// TIA Portal V17 export
// export: Created 2025-03-05T08:02:23.2667087Z, ExportSetting WithDefaults, DisplayName Totally Integrated Automation Portal, DisplayVersion V17 Update 8, DisplayName TIA Portal Openness, DisplayVersion V17 Update 8, DisplayName TIA Portal Version Control Interface, DisplayVersion V17, DisplayName SINAMICS Startdrive Advanced, DisplayVersion V17 SP2, DisplayName SINAMICS Startdrive G110M, G120, G120C, G120D, G120P, G115D, DisplayVersion V17 SP2, DisplayName SINAMICS Startdrive G130, G150, S120, S150, SINAMICS MV, S210, DisplayVersion V17 SP2, DisplayName STEP 7 Professional, DisplayVersion V17 Update 8, DisplayName SINUMERIK ONE STEP 7 Toolbox, DisplayVersion V17 Update 12, DisplayName SINUMERIK 840D sl STEP 7 Toolbox, DisplayVersion V17 Update 12, DisplayName STEP 7 Safety, DisplayVersion V17 Update 6, DisplayName WinCC Advanced, DisplayVersion V17 Update 8
TYPE "LAYOUT"
// stored: IsFailsafeCompliant false
   STRUCT
      Arrow : Array[0..79] of Bool;   // Arrow
      LED : Array[0..79] of Bool;   // LED
      Image : Array[0..79] of Bool;   // Image
      Text : Array[0..79] of Bool;   // Text
      IO_field : Array[0..79] of Bool;   // IO_field
      ProgressBar : Array[0..79] of Bool;   // ProgressBar
      Table0 : Bool;   // Table0
      Table1 : Bool;   // Table1
      Table2 : Bool;   // Table2
      Table3 : Bool;   // Table3
      Table4 : Bool;   // Table4
      Table5 : Bool;   // Table5
      Table6 : Bool;   // Table6
      Table7 : Bool;   // Table7
      Curve0 : Bool;   // Curve0
      Curve1 : Bool;   // Curve1
      Curve2 : Bool;   // Curve2
      Curve3 : Bool;   // Curve3
      Curve4 : Bool;   // Curve4
      Curve5 : Bool;   // Curve5
      Curve6 : Bool;   // Curve6
      Curve7 : Bool;   // Curve7
      Internet0 : Bool;   // Internet0
      Internet1 : Bool;   // Internet1
      Internet2 : Bool;   // Internet2
      Internet3 : Bool;   // Internet3
      Internet4 : Bool;   // Internet4
      Internet5 : Bool;   // Internet5
      Internet6 : Bool;   // Internet6
      Internet7 : Bool;   // Internet7
      SoftkeyLeft0 : Bool;   // SoftkeyLeft0
      SoftkeyLeft1 : Bool;   // SoftkeyLeft1
      SoftkeyLeft2 : Bool;   // SoftkeyLeft2
      SoftkeyLeft3 : Bool;   // SoftkeyLeft3
      SoftkeyLeft4 : Bool;   // SoftkeyLeft4
      SoftkeyLeft5 : Bool;   // SoftkeyLeft5
      SoftkeyLeftAll : Bool;   // SoftkeyLeftAll
      reserveleft : Bool;   // reserveleft
      SoftkeyRight0 : Bool;   // SoftkeyRight0
      SoftkeyRight1 : Bool;   // SoftkeyRight1
      SoftkeyRight2 : Bool;   // SoftkeyRight2
      SoftkeyRight3 : Bool;   // SoftkeyRight3
      SoftkeyRight4 : Bool;   // SoftkeyRight4
      SoftkeyRight5 : Bool;   // SoftkeyRight5
      SoftkeyRightAll : Bool;   // SoftkeyRightAll
      reserveright : Bool;   // reserveright
      Pushbutton0 : Bool;   // Pushbutton0
      Pushbutton1 : Bool;   // Pushbutton1
      Pushbutton2 : Bool;   // Pushbutton2
      Pushbutton3 : Bool;   // Pushbutton3
      Pushbutton4 : Bool;   // Pushbutton4
      Pushbutton5 : Bool;   // Pushbutton5
      Pushbutton6 : Bool;   // Pushbutton6
      Pushbutton7 : Bool;   // Pushbutton7
      Pushbutton8 : Bool;   // Pushbutton8
      Pushbutton9 : Bool;   // Pushbutton9
      Pushbutton10 : Bool;   // Pushbutton10
      Pushbutton11 : Bool;   // Pushbutton11
      Pushbutton12 : Bool;   // Pushbutton12
      Pushbutton13 : Bool;   // Pushbutton13
      Pushbutton14 : Bool;   // Pushbutton14
      Pushbutton15 : Bool;   // Pushbutton15
      Pushbutton16 : Bool;   // Pushbutton16
      Pushbutton17 : Bool;   // Pushbutton17
      Pushbutton18 : Bool;   // Pushbutton18
      Pushbutton19 : Bool;   // Pushbutton19
      Pushbutton20 : Bool;   // Pushbutton20
      Pushbutton21 : Bool;   // Pushbutton21
      Pushbutton22 : Bool;   // Pushbutton22
      Pushbutton23 : Bool;   // Pushbutton23
      Pushbutton24 : Bool;   // Pushbutton24
      Pushbutton25 : Bool;   // Pushbutton25
      Pushbutton26 : Bool;   // Pushbutton26
      Pushbutton27 : Bool;   // Pushbutton27
      Pushbutton28 : Bool;   // Pushbutton28
      Pushbutton29 : Bool;   // Pushbutton29
      Pushbutton30 : Bool;   // Pushbutton30
      Pushbutton31 : Bool;   // Pushbutton31
      byte69 : Byte;   // byte69
   END_STRUCT;
END_TYPE
